FUNCTION_BLOCK FB_CsvPersistentEventStorage IMPLEMENTS I_PersistentEventStorage
VAR
	fbFileOpen : FB_FileOpen := (sPathName := 'C:\ Events.log' , nMode :=  FOPEN_MODEAPPEND OR FOPEN_MODETEXT ) ;
	fbFilePuts  : FB_FilePuts ;
	fbFileClose : Fb_FileClose ;
	eWriteState : (FILE_OPEN_TRIGGER ,FILE_OPEN , WAIT_FOR_EVENT, WRITE_EVENT_TRIGGER, WRITE_EVENT,FILE_CLOSE_TRIGGER, FILE_CLOSE, ERROR ) ;
	StEventWrittenToFile : St_Event ;
	
	CsvString : T_MaxString ;
	FILE_CLOSE_TRIGGER :INT ;
END_VAR


CASE eWriteState OF
	
	FILE_OPEN_TRIGGER:
		fbFileOpen(bExecute := TRUE ) ;
		eWriteState := FILE_OPEN ;
		
		
	FILE_OPEN 		:
		fbFileOpen(bExecute := FALSE ) ;
		IF fbFileOpen.bError THEN
			eWriteState := ERROR ;
		ELSIF NOT fbFileOpen.bBusy AND fbFileOpen.hFile <> 0 THEN
			eWriteState := WAIT_FOR_EVENT ;	
		END_IF
  	WAIT_FOR_EVENT 	:
	//code yok
	WRITE_EVENT_TRIGGER 	:
		CsvString := CreateCsvString(stEvent := StEventWrittenToFile) ;
		fbFilePuts(bExecute := TRUE,
					sLine := CsvString ,
					hFile := fbFileOpen.hFile) ;
		eWriteState := WRITE_EVENT ;	
		
	WRITE_EVENT 	:
		fbFilePuts(bExecute := FALSE);
		IF fbFilePuts.bError THEN
			eWriteState := ERROR ;
		ELSIF NOT fbFilePuts.bBusy THEN
			eWriteState := WAIT_FOR_EVENT ;
		END_IF
	
	FILE_CLOSE_TRIGGER :
		fbFileClose(bExecute := TRUE ,
				hFile := fbFileOpen.hFile);
		eWriteState := WRITE_EVENT ;
	
	FILE_CLOSE		:
		fbFileClose(bExecute := FALSE ) ;
		IF fbFileClose.bError THEN
			eWriteState := ERROR ;
		ELSIF  NOT fbFileClose.bBusy THEN
			eWriteState := FILE_OPEN_TRIGGER ;
		END_IF
	ERROR :
		//CODE YOK
	
	
END_CASE

METHOD PRIVATE CreateCsvString : T_MaxString
VAR_INPUT
	stEvent : REFERENCE TO ST_EVENt ;
END_VAR
VAR
	TempString : T_MaxString ;
END_VAR
TempString := TO_STRING(stEvent.eEventType) ;
TempString := CONCAT(STR1:= TempString , STR2 := ',') ;
TempString := CONCAT(STR1:= TempString , STR2 := TO_STRING (stEvent.eEventSeverity));
TempString := CONCAT(STR1:= TempString , STR2 := ',') ;
TempString := CONCAT(STR1:= TempString , STR2 := TO_STRING (stEvent.nEventIdentiy )) ;
TempString := CONCAT(STR1:= TempString , STR2 := ',') ;
TempString := CONCAT(STR1:= TempString , STR2 := stEvent.sEventText);
TempString := CONCAT(STR1:= TempString , STR2 := ',') ;
TempString := CONCAT(STR1:= TempString , STR2 := TO_STRING (stEvent.dtTimeStamp)) ;
TempString := CONCAT(STR1:= TempString , STR2 := '$n') ;

CreateCsvString := TempString ;
END_METHOD

{warning 'add method implementation '}
METHOD StoreEvent
VAR_INPUT
	stEvent	: St_Event;
END_VAR
IF eWriteState = WAIT_FOR_EVENT THEN
	eWriteState := Write_EVENT ;
	StEventWrittenToFile := stEvent ;
	
	
END_IF
END_METHOD

END_FUNCTION_BLOCK

(* stored: Version 1.1.0.1, ProductVersion 3.1.4024.12
   POU FB_CsvPersistentEventStorage: Id {7ff528b5-f284-4bd1-89ac-0b897b26279c}, SpecialFunc None
   Method CreateCsvString: Id {0d4cdda5-417b-4e56-bd02-87377824357c}
   Method StoreEvent: Id {9f1377bb-5c1f-4ceb-9d75-a0ce46d8993e} *)
